FUNCTION_BLOCK Load1Check (* Template for a Basic Function Block Type *)
  (* Standard: 61499-2 *)
  (* Version 1.0, 2021-07-29, Tuojian Lyu *)
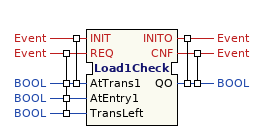
  EVENT_INPUT
    INIT WITH AtTrans1; (* Initialization Request *)
    REQ WITH AtTrans1, AtEntry1, TransLeft; (* Normal Execution Request *)
  END_EVENT
  EVENT_OUTPUT
    INITO WITH QO; (* Initialization Confirm *)
    CNF WITH QO; (* Execution Confirmation *)
  END_EVENT
  VAR_INPUT
    AtTrans1 : BOOL; (* Input event qualifier *)
    AtEntry1 : BOOL;
    TransLeft : BOOL;
  END_VAR
  VAR_OUTPUT
    QO : BOOL; (* Output event qualifier *)
  END_VAR
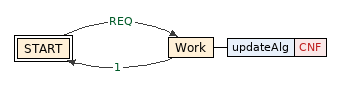
  EC_STATES
    START; (* Initial State *)
    Work : updateAlg -> CNF;
  END_STATES
  EC_TRANSITIONS
    START TO Work := REQ;
    Work TO START := 1;
  END_TRANSITIONS
  ALGORITHM updateAlg IN ST:
IF (TRUE = AtEntry1) AND (FALSE = TransLeft) THEN
QO := TRUE;
END_IF;

IF (TRUE = AtTrans1) AND (FALSE = TransLeft) THEN
QO := TRUE;
END_IF;

IF (FALSE = AtEntry1) AND (FALSE = AtTrans1) THEN
QO := FALSE;
END_IF;
  END_ALGORITHM
END_FUNCTION_BLOCK
